PROGRAM P_HmiHandling
VAR
	ntClosePlcHmi : NT_StartProcess;
	bClose : BOOL := FALSE;
END_VAR


ntClosePlcHmi(
	NETID:='' , 
	PATHSTR:='C:\Windows\System32\cmd.exe' , 
	DIRNAME:='C:\Windows\System32' , 
	COMNDLINE:='/c "C:\HMI\ClosePlcHmi.cmd"' , 
	START:=bClose , 
	TMOUT:=T#5S ,
 
	BUSY=> , 
	ERR=> , 
	ERRID=> );

END_PROGRAM

(* stored: Version 1.1.0.1, ProductVersion 3.1.4024.3
   POU P_HmiHandling: Id {4165462b-3bf4-4761-9d2d-90c8ce86ceb3}, SpecialFunc None *)
